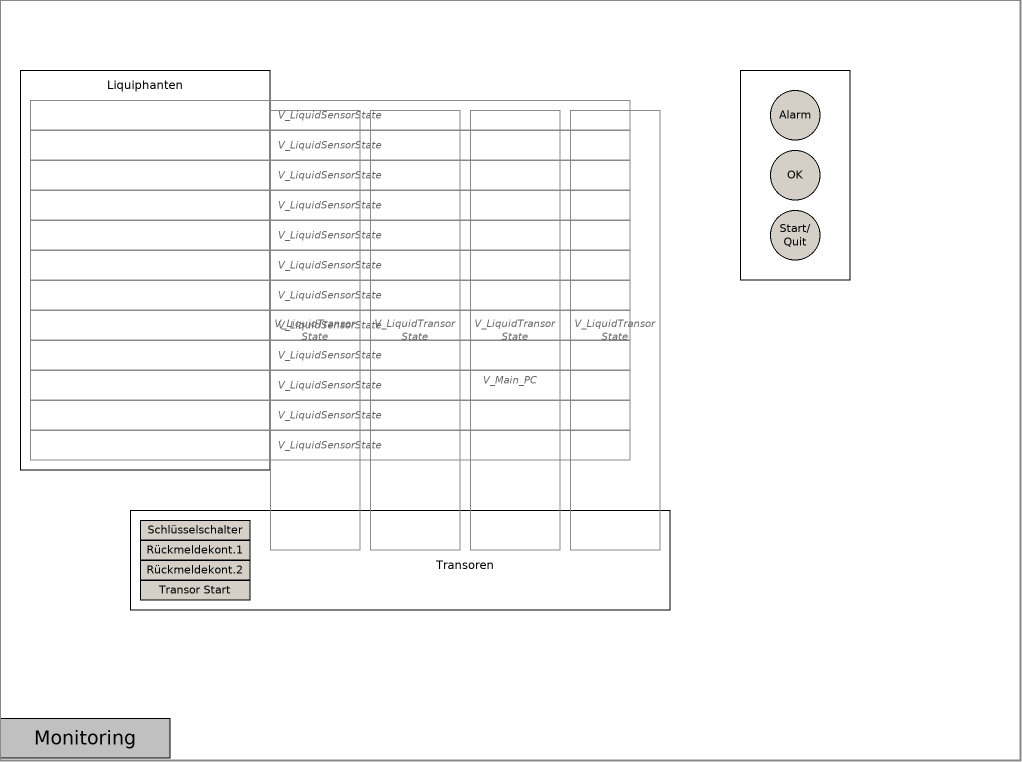
VISUALIZATION V_Monitoring  // 1022x762
    Frame (0,0 1020x760)
        shows V_Main_PC()
    Rectangle (20,70 250x400)
    Rectangle (130,510 540x100)
    Rectangle (0,718 170x40), "Monitoring"
    Frame (30,100 600x30)
        shows V_LiquidSensorState(IOfbLiquidSensor := PLC_PRG.fbLiquidMonitoring.fbLiquidSensor[1])
    Frame (30,130 600x30)
        shows V_LiquidSensorState(IOfbLiquidSensor := PLC_PRG.fbLiquidMonitoring.fbLiquidSensor[2])
    Frame (30,160 600x30)
        shows V_LiquidSensorState(IOfbLiquidSensor := PLC_PRG.fbLiquidMonitoring.fbLiquidSensor[3])
    Frame (30,190 600x30)
        shows V_LiquidSensorState(IOfbLiquidSensor := PLC_PRG.fbLiquidMonitoring.fbLiquidSensor[4])
    Frame (30,220 600x30)
        shows V_LiquidSensorState(IOfbLiquidSensor := PLC_PRG.fbLiquidMonitoring.fbLiquidSensor[5])
    Frame (30,250 600x30)
        shows V_LiquidSensorState(IOfbLiquidSensor := PLC_PRG.fbLiquidMonitoring.fbLiquidSensor[6])
    Frame (30,280 600x30)
        shows V_LiquidSensorState(IOfbLiquidSensor := PLC_PRG.fbLiquidMonitoring.fbLiquidSensor[7])
    Frame (30,310 600x30)
        shows V_LiquidSensorState(IOfbLiquidSensor := PLC_PRG.fbLiquidMonitoring.fbLiquidSensor[8])
    Frame (30,340 600x30)
        shows V_LiquidSensorState(IOfbLiquidSensor := PLC_PRG.fbLiquidMonitoring.fbLiquidSensor[9])
    Frame (30,370 600x30)
        shows V_LiquidSensorState(IOfbLiquidSensor := PLC_PRG.fbLiquidMonitoring.fbLiquidSensor[10])
    Frame (30,400 600x30)
        shows V_LiquidSensorState(IOfbLiquidSensor := PLC_PRG.fbLiquidMonitoring.fbLiquidSensor[11])
    Frame (30,430 600x30)
        shows V_LiquidSensorState(IOfbLiquidSensor := PLC_PRG.fbLiquidMonitoring.fbLiquidSensor[12])
    Frame (270,110 90x440)
        shows V_LiquidTransorState(IOfbTransor := PLC_PRG.fbLiquidMonitoring.fbTransor[1])
    Frame (370,110 90x440)
        shows V_LiquidTransorState(IOfbTransor := PLC_PRG.fbLiquidMonitoring.fbTransor[2])
    Frame (470,110 90x440)
        shows V_LiquidTransorState(IOfbTransor := PLC_PRG.fbLiquidMonitoring.fbTransor[3])
    Frame (570,110 90x440)
        shows V_LiquidTransorState(IOfbTransor := PLC_PRG.fbLiquidMonitoring.fbTransor[4])
    Rectangle (270,550 390x30), "Transoren"
    Rectangle (30,70 230x30), "Liquiphanten"
    Rectangle (740,70 110x210)
    Ellipse (770,90 50x50), "Alarm", colour toggle: PLC_PRG.fbLiquidMonitoring.QbLMStatusAlarm
    Ellipse (770,150 50x50), "OK", colour toggle: PLC_PRG.fbLiquidMonitoring.QbLMStatusOK
    Ellipse (770,210 50x50), "Start/ Quit", tooltip "Alarm quittieren und Transoren starten", colour toggle: PLC_PRG.fbLiquidMonitoring.QbLMStartQuit
        tap PLC_PRG.fbLiquidMonitoring.VbStartQuit
    Rectangle (140,520 110x20), "Schlüsselschalter", colour toggle: PLC_PRG.fbLiquidMonitoring.IbKeySwitch
    Rectangle (140,540 110x20), "Rückmeldekont.1", colour toggle: PLC_PRG.fbLiquidMonitoring.IbContactorResponse1
    Rectangle (140,560 110x20), "Rückmeldekont.2", colour toggle: PLC_PRG.fbLiquidMonitoring.IbContactorResponse2
    Rectangle (140,580 110x20), "Transor Start", colour toggle: PLC_PRG.fbLiquidMonitoring.QbStartTransor
END_VISUALIZATION

(* stored: Version 1.1.0.1, ProductVersion 3.1.4018.10
   Visu V_Monitoring: Id {46b28f1c-aea0-4a4b-8e95-9c92969f139a} *)
